FUNCTION_BLOCK PUBLIC EcMasterDeviceCount IMPLEMENTS IEcTask
VAR_INPUT
END_VAR
VAR_OUTPUT
END_VAR
VAR
	iState : INT;
	masterDeviceCount : Tc2_EtherCAT.FB_EcGetSlaveCount;
	_execute: BOOL;
	_done: BOOL;
	_busy: BOOL;
	_error: BOOL;
	_netId: AMSNETID;
END_VAR

CASE iState OF
	0:
		IF _execute THEN
			_done := FALSE;
			_busy := TRUE;
			_error := FALSE;
			masterDeviceCount.bExecute := TRUE;
			IF masterDeviceCount.bBusy THEN
				iState := 10;
				_execute := false;
			END_IF
		END_IF
	10:
		IF NOT masterDeviceCount.bBusy THEN
			IF NOT masterDeviceCount.bError THEN
				_done := TRUE;
			ELSE
				_error := TRUE;
			END_IF
			_busy := FALSE;
			masterDeviceCount.bExecute := FALSE;
			iState := 0;
		END_IF
END_CASE

masterDeviceCount(sNetId := Tc2_System.F_CreateAmsNetId(nIds := NetId));

{warning 'add method implementation '}
METHOD Abort : BOOL
masterDeviceCount.bExecute := FALSE;
_busy := FALSE;
_execute := FALSE;
Abort := TRUE;
iState := 0;
END_METHOD

{warning 'add property implementation'}
PROPERTY Busy : BOOL
GET
Busy := _busy;
END_GET
END_PROPERTY

{warning 'add property implementation'}
PROPERTY Done : BOOL
GET
Done := _done;
END_GET
END_PROPERTY

{warning 'add property implementation'}
PROPERTY Error : BOOL
GET
Error := _error;
END_GET
END_PROPERTY

METHOD Execute : BOOL
VAR_INPUT
END_VAR
IF NOT Busy THEN
	Execute := _execute := TRUE;
END_IF
END_METHOD

{warning 'add property implementation'}
PROPERTY NetID : amsnetid
GET
NetID := _netId;
END_GET
SET
_netId := NetID;
END_SET
END_PROPERTY

PROPERTY NumberDevices : uint
GET
NumberDevices := masterDeviceCount.nSlaves;
END_GET
END_PROPERTY

END_FUNCTION_BLOCK

(* stored: Version 1.1.0.1, ProductVersion 3.1.4024.11
   POU EcMasterDeviceCount: Id {423676d1-5e98-4b58-aeb3-4d7ba3e75786}, SpecialFunc None
   Method Abort: Id {482aaa32-fc09-4c8e-881c-6eabe1a2e522}
   Property Busy: Id {adc3a81d-2838-47ed-8b19-de9731afa905}
   Get Get: Id {21447dcd-0743-4691-8714-b3a1aa328079}
   Property Done: Id {7fa31933-5ae9-467f-b833-56fbd23c2268}
   Get Get: Id {914ebbda-6f92-4e7e-a4b6-81f919788ff6}
   Property Error: Id {e032720c-e318-4305-b710-f37374dc4e33}
   Get Get: Id {b99db219-4ec2-44f0-bec0-63391aa50bd0}
   Method Execute: Id {6afa2a6b-3b50-4a86-bf47-e3840676a4bd}
   Property NetID: Id {eb8cb74b-4d84-43ef-8c24-8b8a8c2044c2}
   Get Get: Id {7ac222c8-00b1-4eba-b4a7-64ae6c42e1b5}
   Set Set: Id {806a648c-699a-478c-b667-2cb864f4e8f1}
   Property NumberDevices: Id {2a6ef48d-f582-4562-87eb-becb9d375441}
   Get Get: Id {26f117f9-e31c-4f3f-88da-a013bf942179} *)
